FUNCTION_BLOCK D_5States_5Algo (* Basic FB with empty ECC *)
  (* Standard: 61499-2 *)
  (* Version 1.0, 2023-09-22, AK124910 *)
  PACKAGE servSeq;
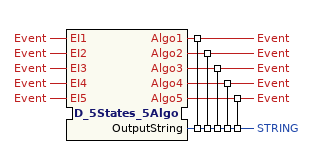
  EVENT_INPUT
    EI1;
    EI2;
    EI3;
    EI4;
    EI5;
  END_EVENT
  EVENT_OUTPUT
    Algo1 WITH OutputString;
    Algo2 WITH OutputString;
    Algo3 WITH OutputString;
    Algo4 WITH OutputString;
    Algo5 WITH OutputString;
  END_EVENT
  VAR_OUTPUT
    OutputString : STRING;
  END_VAR
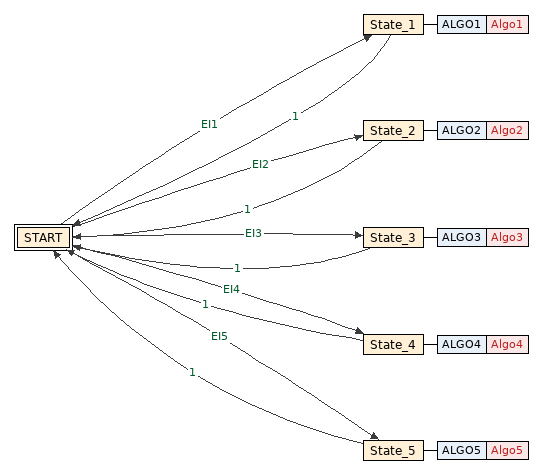
  EC_STATES
    START; (* Initial State *)
    State_1 : ALGO1 -> Algo1;
    State_2 : ALGO2 -> Algo2;
    State_3 : ALGO3 -> Algo3;
    State_4 : ALGO4 -> Algo4;
    State_5 : ALGO5 -> Algo5;
  END_STATES
  EC_TRANSITIONS
    START TO State_1 := EI1;
    State_1 TO START := 1;
    START TO State_2 := EI2;
    State_2 TO START := 1;
    START TO State_3 := EI3;
    State_3 TO START := 1;
    START TO State_4 := EI4;
    State_4 TO START := 1;
    START TO State_5 := EI5;
    State_5 TO START := 1;
  END_TRANSITIONS
  ALGORITHM ALGO1 IN ST:
OutputString := CONCAT(OutputString, 'ALGO1/');
  END_ALGORITHM
  ALGORITHM ALGO2 IN ST:
OutputString := CONCAT(OutputString, 'ALGO2/');
  END_ALGORITHM
  ALGORITHM ALGO3 IN ST:
OutputString := CONCAT(OutputString, 'ALGO3/');
  END_ALGORITHM
  ALGORITHM ALGO4 IN ST:
OutputString := CONCAT(OutputString, 'ALGO4/');
  END_ALGORITHM
  ALGORITHM ALGO5 IN ST:
OutputString := CONCAT(OutputString, 'ALGO5/');
  END_ALGORITHM
END_FUNCTION_BLOCK
